Staubli VAL3: j213_external24V.dtx

mdesc mNomSpeed
dio dDioMainPowerOk = {link=PowerSupplyIO\mainPowerOk}
